(* PLC project Tc2_Utilities.FB_FileRingBuffer Demo, tc3-libraries-kb TwinCAT 3.1 *)
(* stored: creationDateTime 2026-05-10T20:00:00, modificationDateTime 2026-05-10T20:00:00 *)

PROGRAM P_Demo_FB_FileRingBuffer
  VAR
    fbFB_FileRingBuffer : FB_FileRingBuffer;  (* Tc2_Utilities.FB_FileRingBuffer 实例 *)
    arg_sNetId : T_AmsNetId;  (* VAR_INPUT sNetId *)
    arg_sPathName : T_MaxString;  (* VAR_INPUT sPathName *)
    arg_ePath : E_OpenPath;  (* VAR_INPUT ePath *)
    arg_nID : UDINT;  (* VAR_INPUT nID *)
    arg_cbBuffer : UDINT;  (* VAR_INPUT cbBuffer *)
    arg_bOverwrite : BOOL;  (* VAR_INPUT bOverwrite *)
    arg_pWriteBuff : POINTER TO BYTE;  (* VAR_INPUT pWriteBuff *)
    arg_cbWriteLen : UDINT;  (* VAR_INPUT cbWriteLen *)
    arg_pReadBuff : POINTER TO BYTE;  (* VAR_INPUT pReadBuff *)
    arg_cbReadLen : UDINT;  (* VAR_INPUT cbReadLen *)
    arg_tTimeout : TIME;  (* VAR_INPUT tTimeout *)
    out_bBusy : BOOL;  (* VAR_OUTPUT bBusy *)
    out_bError : BOOL;  (* VAR_OUTPUT bError *)
    out_nErrId : UDINT;  (* VAR_OUTPUT nErrId *)
    out_cbReturn : UDINT;  (* VAR_OUTPUT cbReturn *)
    out_stHeader : ST_FileRBufferHead;  (* VAR_OUTPUT stHeader *)
  END_VAR

            // ============================================================
// Tc2_Utilities.FB_FileRingBuffer 演示程序（FB 实例）
// ============================================================
// 验证步骤：
//   1. 引用 Tc2_Utilities（及依赖类型所在库 Tc2_System 等）
//   2. 编译 + 登录
//   3. 按 doc.md 给 arg_* 赋值
//   4. 在线监视 out_* / io_* 输出
// ============================================================

fbFB_FileRingBuffer(
    sNetId := arg_sNetId,
    sPathName := arg_sPathName,
    ePath := arg_ePath,
    nID := arg_nID,
    cbBuffer := arg_cbBuffer,
    bOverwrite := arg_bOverwrite,
    pWriteBuff := arg_pWriteBuff,
    cbWriteLen := arg_cbWriteLen,
    pReadBuff := arg_pReadBuff,
    cbReadLen := arg_cbReadLen,
    tTimeout := arg_tTimeout,
    bBusy => out_bBusy,
    bError => out_bError,
    nErrId => out_nErrId,
    cbReturn => out_cbReturn,
    stHeader => out_stHeader
);

          
END_PROGRAM
